(* CODESYS project Project.project

Project tree, tasks and I/O mapping:
  Device : CODESYS Control Win V3, 3S - Smart Software Solutions GmbH, version 3.5.3.50
    application Application
      libraries: Standard, 3.5.2.0 (System); VisuDialogs, * (System)
      task MainTask (cyclic, interval t#20ms, priority 1) calls PLC_PRG, Simulation
      task VISU_TASK (cyclic, interval 100 ms, priority 30) calls VisuElems.Visu_Prg
      program PLC_PRG [SFC]: T5s, T2s, T3s, Initialize, checkiffull, nextbottle, deactivateStart
      global variables GVL
      program Simulation [ST]
      visualisation Visualization
  text list GlobalTextList
  GlobalImagePool
*)

// Device/Application/GVL
VAR_GLOBAL
END_VAR
VAR_GLOBAL
	start: BOOL;
	motor: BOOL;
	f1: BOOL;
	f2: BOOL;
	f3: BOOL;
	pos_bottle: INT := 0;
	counter: INT := 0;
	fialesmax: INT := 500;
	fiales: LREAL := 500;
	stop: BOOL;
	next_bottle: BOOL;
	save: BOOL;
	stop1: BOOL;
	maxperday: INT;
	bell: BOOL;
END_VAR

// Device/Application/PLC_PRG
PROGRAM PLC_PRG
VAR
	Timer: TIME;
	TP_0: TP;
	TON_0: TON;
	TP_time3: TIME;
	TP_time5: TIME;
	TP_time2: TIME;
	start_timer1: BOOL;
	start_timer2: BOOL;
	start_timer3: BOOL;
	T5: TIME := T#5s;
	T3: TIME := T#3s;
	T2: TIME := T#2S;
END_VAR
VAR_INPUT
	
	SFCPause: BOOL;
END_VAR

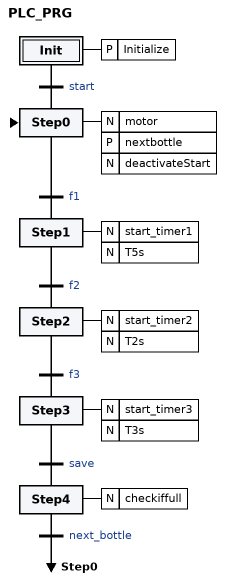
INITIAL_STEP Init:
    Initialize(P);
END_STEP
TRANSITION FROM Init TO Step0
    := start;
END_TRANSITION
STEP Step0:
    motor(N);
    nextbottle(P);
    deactivateStart(N);
END_STEP
TRANSITION FROM Step0 TO Step1
    := f1;
END_TRANSITION
STEP Step1:
    start_timer1(N);
    T5s(N);
END_STEP
TRANSITION FROM Step1 TO Step2
    := f2;
END_TRANSITION
STEP Step2:
    start_timer2(N);
    T2s(N);
END_STEP
TRANSITION FROM Step2 TO Step3
    := f3;
END_TRANSITION
STEP Step3:
    start_timer3(N);
    T3s(N);
END_STEP
TRANSITION FROM Step3 TO Step4
    := save;
END_TRANSITION
STEP Step4:
    checkiffull(N);
END_STEP
TRANSITION FROM Step4 TO Step0
    := next_bottle;
END_TRANSITION

ACTION T5s:
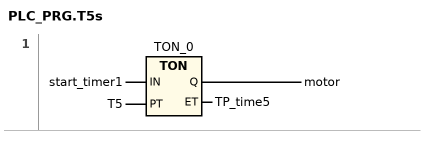
// NETWORK 1
TON_0(IN := start_timer1, PT := T5, ET => TP_time5); // TON
motor := TON_0.Q;
END_ACTION

ACTION T2s:
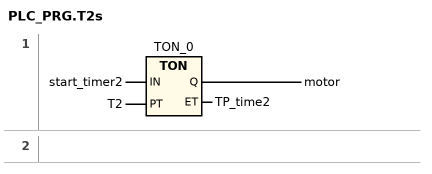
// NETWORK 1
TON_0(IN := start_timer2, PT := T2, ET => TP_time2); // TON
motor := TON_0.Q;

// NETWORK 2
END_ACTION

ACTION T3s:
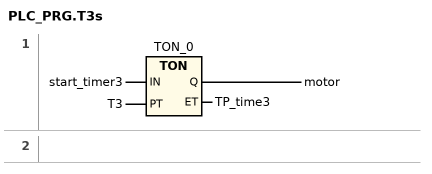
// NETWORK 1
TON_0(IN := start_timer3, PT := T3, ET => TP_time3); // TON
motor := TON_0.Q;

// NETWORK 2
END_ACTION

ACTION Initialize:
motor:=FALSE;
start:=FALSE;
counter:=0;
pos_bottle:=0;
f1:=FALSE;
f2:=FALSE;
f3:=FALSE;
bell:=FALSE;
END_ACTION

ACTION checkiffull:
save:=FALSE;

IF (counter>fialesmax OR fiales<0 OR counter>(maxperday-1)) THEN
	motor:=FALSE;
	next_bottle:=FALSE;
	bell:=TRUE;
ELSE
	next_bottle:=TRUE;
END_IF
END_ACTION

ACTION nextbottle:
next_bottle:=FALSE;
fiales:=fiales-0.5;
bell:=FALSE;
END_ACTION

ACTION deactivateStart:
stop1:=FALSE;
start:=FALSE;
END_ACTION

END_PROGRAM

// Device/Application/Simulation
PROGRAM Simulation

VAR_INPUT
	
	
END_VAR
VAR
	temp: BOOL;
	temp3: BOOL;
	temp2: BOOL;
	temp1: BOOL;
END_VAR



IF motor THEN
	pos_bottle:=pos_bottle+1;
END_IF;

IF (pos_bottle>=145 AND pos_bottle<=155 AND NOT(stop)) THEN
	f1:=TRUE;
	temp1:=f1;	
	motor:=FALSE;
ELSE
	f1:=FALSE;
END_IF;

IF (pos_bottle>=295 AND pos_bottle<=305 AND NOT(stop)) THEN
	f2:=TRUE;
	temp2:=f2;
	motor:=FALSE;
ELSE
	f2:=FALSE;
END_IF;

IF (pos_bottle>=445 AND pos_bottle<=455 AND NOT(stop)) THEN
	f3:=TRUE;
	temp3:=f3;
	motor:=FALSE;
ELSE
	f3:=FALSE;
END_IF;

IF (pos_bottle>595) THEN
	
	counter:=counter+1;
	pos_bottle:=0;
	save:=TRUE;
END_IF

IF (stop) THEN
	PLC_PRG.SFCPause:=TRUE;
	f1:=f2:=f3:=FALSE;
	motor:=FALSE;
	stop1:=TRUE;
	stop:=FALSE;
	ELSE
	    IF (start)	THEN
          PLC_PRG.SFCPause:=FALSE;
		  start:=false;
	    END_IF    
END_IF

END_PROGRAM

// Device/Application/Visualization
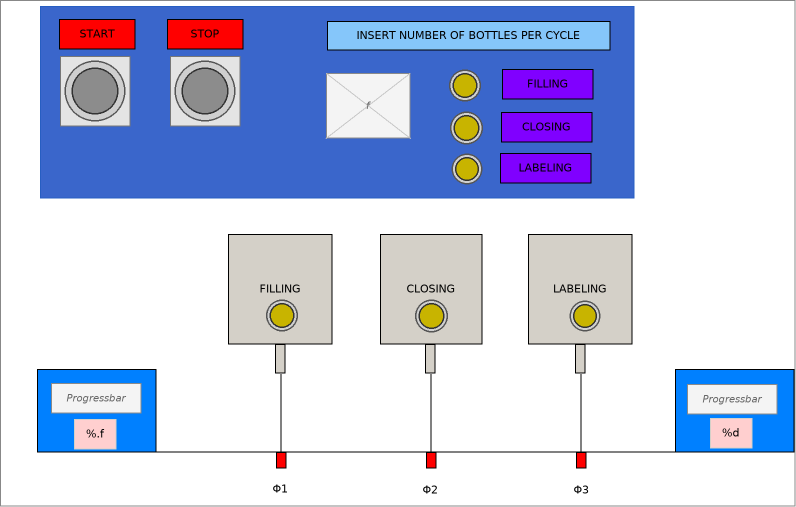
VISUALIZATION Visualization  // 796x507
    RoundedRectangle (40,6 594x192)
    Image (124,380 22x72), image: reusing-plastic-bottle
        p3560616238: pos_bottle
    PushSwitch (60,56 70x70), variable: start, behaviour: TOGGLE, style: Switch-PushSwitch-Gray
    PushSwitch (170,56 70x70), variable: stop, behaviour: TOGGLE, style: Switch-PushSwitch-Gray
    Line (128,452)
    Line (790,452) (129,452)
    Rectangle (37,369 119x83)
    Rectangle (675,369 119x83)
    RoundedRectangle (228,234 104x110), "FILLING"
    Rectangle (275,344 10x29)
    Rectangle (425,344 10x29)
    RoundedRectangle (380,234 102x110), "CLOSING"
    Rectangle (575,344 10x29)
    RoundedRectangle (528,234 104x110), "LABELING"
    Progressbar (687,384 90x30), variable: counter
    Lamp1 (263,297 38x37), variable: f1, style: Lamp-Lamp1-Yellow
    Lamp1 (411,297 41x38), variable: f2, style: Lamp-Lamp1-Yellow
    Lamp1 (565,298 40x36), variable: f3, style: Lamp-Lamp1-Yellow
    Progressbar (51,383 90x30), variable: fiales
    Rectangle (276,452 10x16), colour toggle: f1
    Rectangle (426,452 10x16), colour toggle: f2
    Rectangle (576,452 10x16), colour toggle: f3
    Label (266,474 29x30), "Φ1"
    Label (416,475 29x30), "Φ2"
    Label (567,475 29x30), "Φ3"
    RoundedRectangle (59,19 76x30), "START", colour toggle: start
    RoundedRectangle (167,19 76x30), "STOP", colour toggle: stop
    Line (281,451) (281,374), colour toggle: f1
    Line (431,451) (431,374), colour toggle: f2
    Line (581,451) (581,374), colour toggle: f3
    Textfield (710,418 42x30), "%d", text variable: counter
    Textfield (74,419 42x30), "%.f", text variable: fiales
    RoundedRectangle (327,21 283x29), "INSERT NUMBER OF BOTTLES PER CYCLE"
        OnMouseDown: write maxperday via VisuDialogs.Numpad, min 100, max 999
    Image (326,73 84x65), invisible if: not(bell), image: f
    Lamp1 (446,109 41x38), variable: f2, style: Lamp-Lamp1-Yellow
    Lamp1 (446,67 38x37), variable: f1, style: Lamp-Lamp1-Yellow
    Lamp1 (447,151 40x36), variable: f3, style: Lamp-Lamp1-Yellow
    Textfield (502,69 91x30), "FILLING"
    Textfield (501,112 91x30), "CLOSING"
    Textfield (500,153 91x30), "LABELING"
END_VISUALIZATION
